(* PLC project Untitled1, Beckhoff Automation GmbH TF6420 Database Server Query Analyser 1.0.0.0 *)
(* stored: creationDateTime 2020-05-16T16:04:40, modificationDateTime 2020-05-16T16:04:40 *)

TYPE ST_SelectStruct : STRUCT
  PCB_Number : INT;
  DateTime : DT;
  Free_from_defects : STRING(255);
  M_Point_1 : STRING(255);
  M_Point_1_result : LREAL;
  M_Point_1_reference : DINT;
  M_Point_1_toleracne : DINT;
END_STRUCT;
END_TYPE
